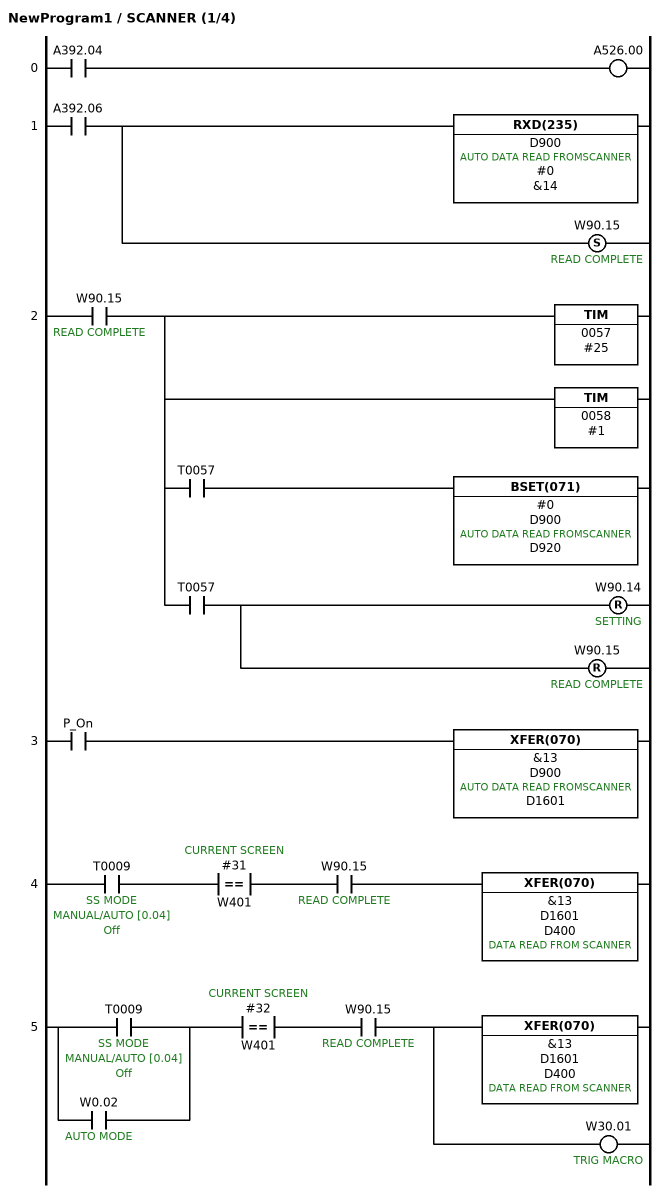
; [picture p24: NewProgram1 / SCANNER, rungs 0-5]
; rung 0
LD A392.04
OUT A526.00
; rung 1
LD A392.06
RXD(235) D900 #0 &14  ; AUTO DATA READ FROMSCANNER
SET W90.15  ; READ COMPLETE
; rung 2
LD W90.15  ; READ COMPLETE
OUT TR0
TIM 0057 #25
TIM 0058 #1
AND T0057
BSET(071) #0 D900 D920  ; AUTO DATA READ FROMSCANNER
LD TR0
AND T0057
RSET W90.14  ; SETTING
RSET W90.15  ; READ COMPLETE
; rung 3
LD P_On
XFER(070) &13 D900 D1601  ; AUTO DATA READ FROMSCANNER
; rung 4
LD T0009  ; SS MODE MANUAL/AUTO [0.04] Off
AND=(300) #31 W401  ; CURRENT SCREEN
AND W90.15  ; READ COMPLETE
XFER(070) &13 D1601 D400  ; DATA READ FROM SCANNER
; rung 5
LD T0009  ; SS MODE MANUAL/AUTO [0.04] Off
OR W0.02  ; AUTO MODE
AND=(300) #32 W401  ; CURRENT SCREEN
AND W90.15  ; READ COMPLETE
XFER(070) &13 D1601 D400  ; DATA READ FROM SCANNER
OUT W30.01  ; TRIG MACRO

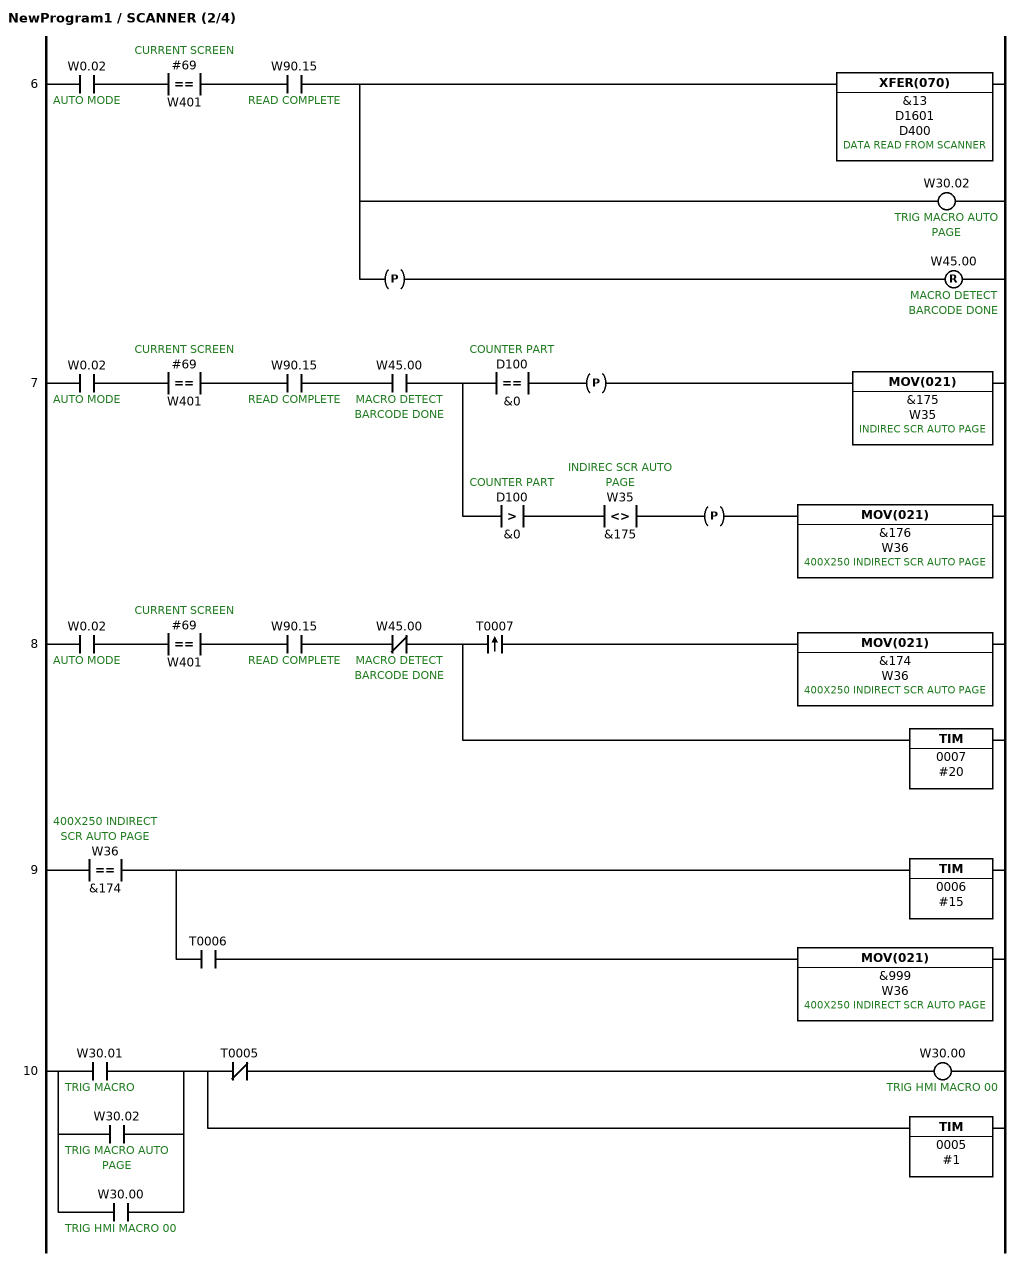
; rung 6
LD W0.02  ; AUTO MODE
AND=(300) #69 W401  ; CURRENT SCREEN
AND W90.15  ; READ COMPLETE
XFER(070) &13 D1601 D400  ; DATA READ FROM SCANNER
OUT W30.02  ; TRIG MACRO AUTO PAGE
UP(521)
RSET W45.00  ; MACRO DETECT BARCODE DONE
; rung 7
LD W0.02  ; AUTO MODE
AND=(300) #69 W401  ; CURRENT SCREEN
AND W90.15  ; READ COMPLETE
AND W45.00  ; MACRO DETECT BARCODE DONE
OUT TR0
AND=(300) D100 &0  ; COUNTER PART
UP(521)
MOV(021) &175 W35  ; INDIREC SCR AUTO PAGE
LD TR0
AND>(320) D100 &0  ; COUNTER PART
AND<>(305) W35 &175  ; INDIREC SCR AUTO PAGE
UP(521)
MOV(021) &176 W36  ; 400X250 INDIRECT SCR AUTO PAGE
; rung 8
LD W0.02  ; AUTO MODE
AND=(300) #69 W401  ; CURRENT SCREEN
AND W90.15  ; READ COMPLETE
ANDNOT W45.00  ; MACRO DETECT BARCODE DONE
OUT TR0
@AND T0007
MOV(021) &174 W36  ; 400X250 INDIRECT SCR AUTO PAGE
LD TR0
TIM 0007 #20
; rung 9
LD=(300) W36 &174  ; 400X250 INDIRECT SCR AUTO PAGE
TIM 0006 #15
AND T0006
MOV(021) &999 W36  ; 400X250 INDIRECT SCR AUTO PAGE
; rung 10
LD W30.01  ; TRIG MACRO
OR W30.02  ; TRIG MACRO AUTO PAGE
OR W30.00  ; TRIG HMI MACRO 00
OUT TR0
ANDNOT T0005
OUT W30.00  ; TRIG HMI MACRO 00
LD TR0
TIM 0005 #1

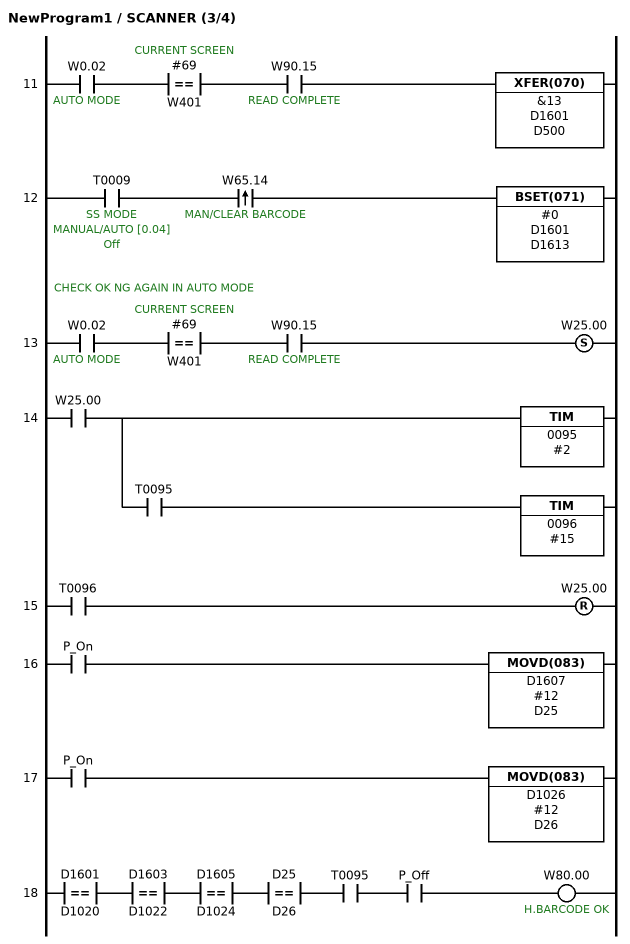
; rung 11
LD W0.02  ; AUTO MODE
AND=(300) #69 W401  ; CURRENT SCREEN
AND W90.15  ; READ COMPLETE
XFER(070) &13 D1601 D500
; rung 12
LD T0009  ; SS MODE MANUAL/AUTO [0.04] Off
@AND W65.14  ; MAN/CLEAR BARCODE
BSET(071) #0 D1601 D1613
; rung 13: CHECK OK NG AGAIN IN AUTO MODE
LD W0.02  ; AUTO MODE
AND=(300) #69 W401  ; CURRENT SCREEN
AND W90.15  ; READ COMPLETE
SET W25.00
; rung 14
LD W25.00
TIM 0095 #2
AND T0095
TIM 0096 #15
; rung 15
LD T0096
RSET W25.00
; rung 16
LD P_On
MOVD(083) D1607 #12 D25
; rung 17
LD P_On
MOVD(083) D1026 #12 D26
; rung 18
LD=L(301) D1601 D1020
AND=L(301) D1603 D1022
AND=L(301) D1605 D1024
AND=(300) D25 D26
AND T0095
AND P_Off
OUT W80.00  ; H.BARCODE OK

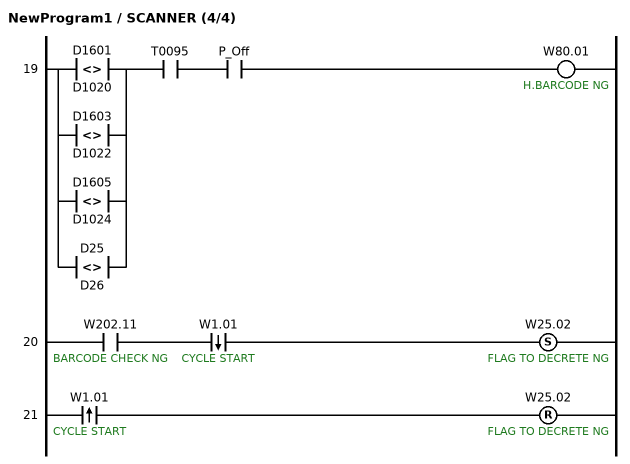
; rung 19
LD<>L(306) D1601 D1020
OR<>L(306) D1603 D1022
OR<>L(306) D1605 D1024
OR<>(305) D25 D26
AND T0095
AND P_Off
OUT W80.01  ; H.BARCODE NG
; rung 20
LD W202.11  ; BARCODE CHECK NG
%AND W1.01  ; CYCLE START
SET W25.02  ; FLAG TO DECRETE NG
; rung 21
@LD W1.01  ; CYCLE START
RSET W25.02  ; FLAG TO DECRETE NG

### Section RFID

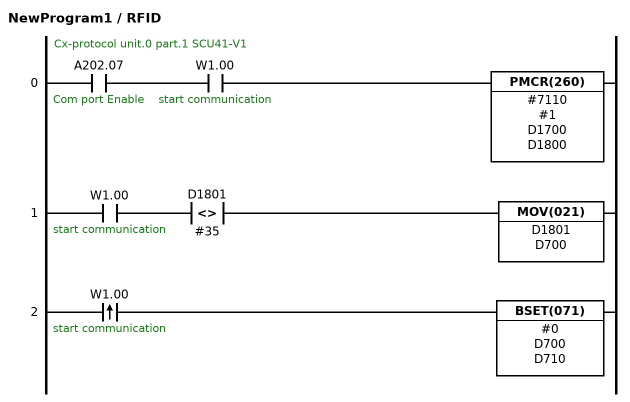
; rung 0: Cx-protocol unit.0 part.1 SCU41-V1
LD A202.07  ; Com port Enable
AND W1.00  ; start communication
PMCR(260) #7110 #1 D1700 D1800
; rung 1
LD W1.00  ; start communication
AND<>(305) D1801 #35
MOV(021) D1801 D700
; rung 2
@LD W1.00  ; start communication
BSET(071) #0 D700 D710

### Section COLORDETECTION

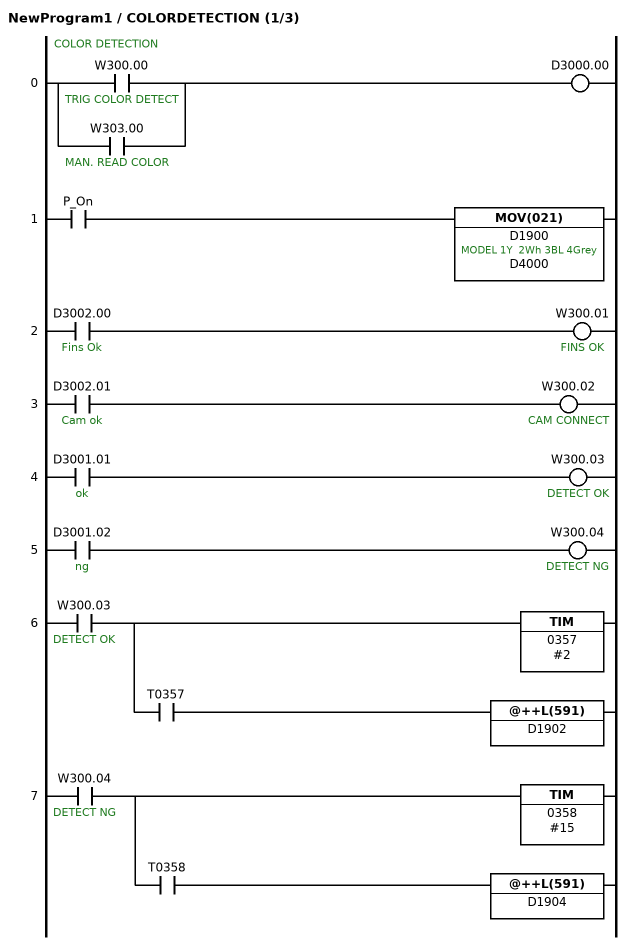
; rung 0: COLOR DETECTION
LD W300.00  ; TRIG COLOR DETECT
OR W303.00  ; MAN. READ COLOR
OUT D3000.00
; rung 1
LD P_On
MOV(021) D1900 D4000  ; MODEL 1Y  2Wh 3BL 4Grey
; rung 2
LD D3002.00  ; Fins Ok
OUT W300.01  ; FINS OK
; rung 3
LD D3002.01  ; Cam ok
OUT W300.02  ; CAM CONNECT
; rung 4
LD D3001.01  ; ok
OUT W300.03  ; DETECT OK
; rung 5
LD D3001.02  ; ng
OUT W300.04  ; DETECT NG
; rung 6
LD W300.03  ; DETECT OK
TIM 0357 #2
AND T0357
@++L(591) D1902
; rung 7
LD W300.04  ; DETECT NG
TIM 0358 #15
AND T0358
@++L(591) D1904

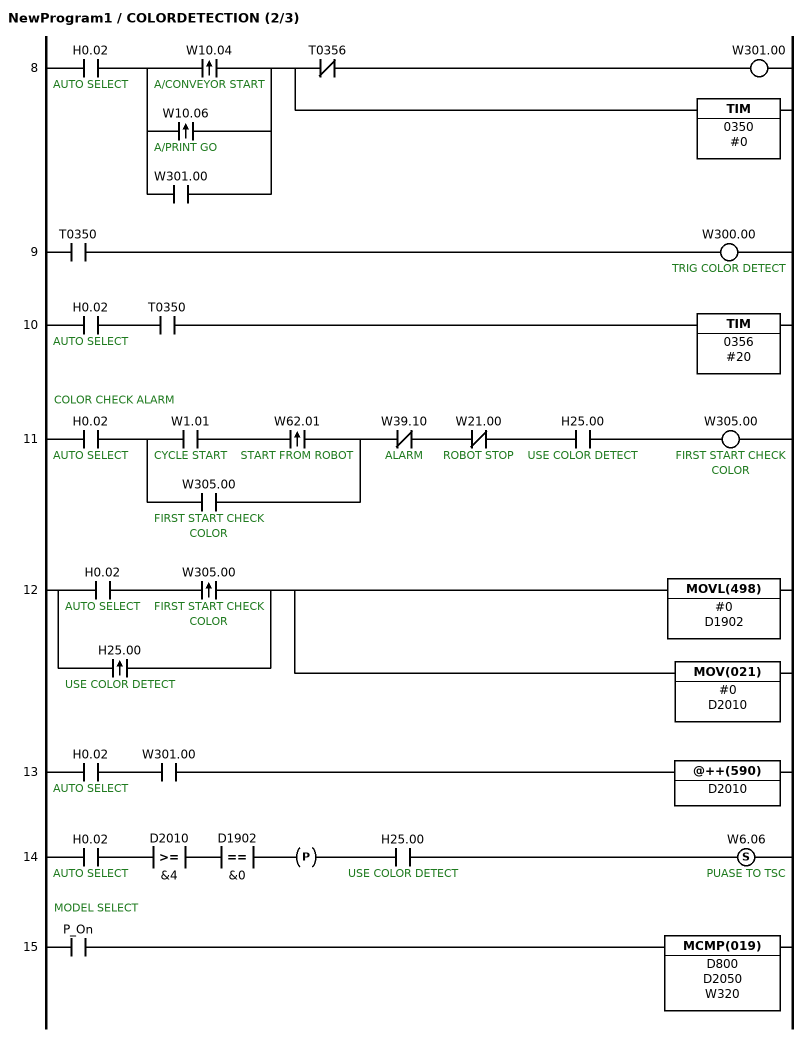
; rung 8
LD H0.02  ; AUTO SELECT
@LD W10.04  ; A/CONVEYOR START
@OR W10.06  ; A/PRINT GO
OR W301.00
ANDLD
OUT TR0
ANDNOT T0356
OUT W301.00
LD TR0
TIM 0350 #0
; rung 9
LD T0350
OUT W300.00  ; TRIG COLOR DETECT
; rung 10
LD H0.02  ; AUTO SELECT
AND T0350
TIM 0356 #20
; rung 11: COLOR CHECK ALARM
LD H0.02  ; AUTO SELECT
LD W1.01  ; CYCLE START
@AND W62.01  ; START FROM ROBOT
OR W305.00  ; FIRST START CHECK COLOR
ANDLD
ANDNOT W39.10  ; ALARM
ANDNOT W21.00  ; ROBOT STOP
AND H25.00  ; USE COLOR DETECT
OUT W305.00  ; FIRST START CHECK COLOR
; rung 12
LD H0.02  ; AUTO SELECT
@AND W305.00  ; FIRST START CHECK COLOR
@OR H25.00  ; USE COLOR DETECT
MOVL(498) #0 D1902
MOV(021) #0 D2010
; rung 13
LD H0.02  ; AUTO SELECT
AND W301.00
@++(590) D2010
; rung 14
LD H0.02  ; AUTO SELECT
AND>=(325) D2010 &4
AND=L(301) D1902 &0
UP(521)
AND H25.00  ; USE COLOR DETECT
SET W6.06  ; PUASE TO TSC
; rung 15: MODEL SELECT
LD P_On
MCMP(019) D800 D2050 W320

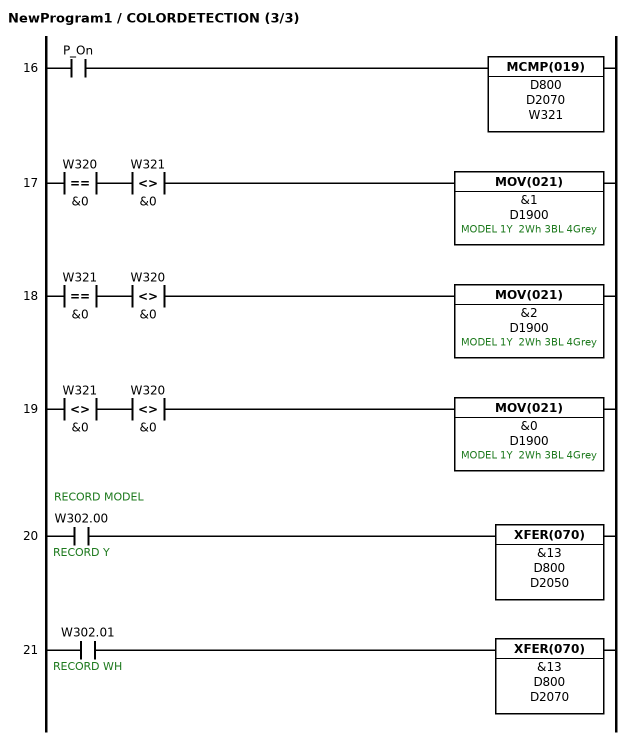
; rung 16
LD P_On
MCMP(019) D800 D2070 W321
; rung 17
LD=(300) W320 &0
AND<>(305) W321 &0
MOV(021) &1 D1900  ; MODEL 1Y  2Wh 3BL 4Grey
; rung 18
LD=(300) W321 &0
AND<>(305) W320 &0
MOV(021) &2 D1900  ; MODEL 1Y  2Wh 3BL 4Grey
; rung 19
LD<>(305) W321 &0
AND<>(305) W320 &0
MOV(021) &0 D1900  ; MODEL 1Y  2Wh 3BL 4Grey
; rung 20: RECORD MODEL
LD W302.00  ; RECORD Y
XFER(070) &13 D800 D2050
; rung 21
LD W302.01  ; RECORD WH
XFER(070) &13 D800 D2070

### Section END
; rung 0
END(001)